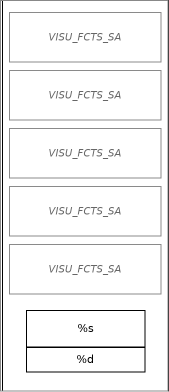
VISUALIZATION VISU_AXE_STD1_FCT_OP_OSC  // 169x392
VAR_IN_OUT
	m_Input_MOTEUR: BLOCK_AXE_STD1_OSCILLANT;
	m_Input_PRG_MOUVEMENT_PS: BLOCK_PRG_MOUVEMENT_PS;
END_VAR
VAR_INPUT
	m_Input_INDEX_MOTEUR : INT;
END_VAR
    RoundedRectangle (2,-1 167x392)
    Rectangle (26,310 119x37), "%s", invisible if: NOT m_Input_PRG_MOUVEMENT_PS.CONF_Balayage[m_Input_INDEX_MOTEUR], text list: 'TextList_Moteurs', text index: 3
    Rectangle (26,347 119x25), "%d", text variable: m_Input_MOTEUR.STATE_NBal, invisible if: NOT m_Input_PRG_MOUVEMENT_PS.CONF_Balayage[m_Input_INDEX_MOTEUR]
    Frame (9,12 152x50)
        shows VISU_FCTS_SA(m_Input_ID_XML := 6, m_Input_Operation := m_Input_MOTEUR.OP_Validation, m_Input_UserRight := PRG_USER.ACTU_USER.FONCTION_SA)
    Frame (9,70 152x50)
        shows VISU_FCTS_SA(m_Input_ID_XML := 7, m_Input_Operation := m_Input_MOTEUR.OP_Stop, m_Input_UserRight := PRG_USER.ACTU_USER.FONCTION_SA)
    Frame (9,128 152x50), invisible if: NOT m_Input_PRG_MOUVEMENT_PS.CONF_Positionnement[m_Input_INDEX_MOTEUR]
        shows VISU_FCTS_SA(m_Input_ID_XML := 8, m_Input_Operation := m_Input_MOTEUR.OP_Position, m_Input_UserRight := PRG_USER.ACTU_USER.FONCTION_SA)
    Frame (9,186 152x50), invisible if: NOT m_Input_PRG_MOUVEMENT_PS.CONF_Rotation[m_Input_INDEX_MOTEUR]
        shows VISU_FCTS_SA(m_Input_ID_XML := 15, m_Input_Operation := m_Input_MOTEUR.OP_Rotation, m_Input_UserRight := PRG_USER.ACTU_USER.FONCTION_SA)
    Frame (9,244 152x50), invisible if: NOT m_Input_PRG_MOUVEMENT_PS.CONF_Balayage[m_Input_INDEX_MOTEUR]
        shows VISU_FCTS_SA(m_Input_ID_XML := 16, m_Input_Operation := m_Input_MOTEUR.OP_Balayage, m_Input_UserRight := PRG_USER.ACTU_USER.FONCTION_SA)
END_VISUALIZATION

(* stored: Version 1.1.0.1, ProductVersion 3.1.4024.10
   Visu VISU_AXE_STD1_FCT_OP_OSC: Id {d1b22bdf-2218-4bf9-806e-eade26dbbb12} *)
